Staubli VAL3: findItem.pgx

public program findItem(InstrItem x_iItem, num& x_nResult)
  local num i
  local num l_nSize
  local num j
  local string l_sItem
  local string l_sMessage
  local num l_nResult
  local bool l_bFound
  local InstrItem l_iInstr[3]
  local string l_sSession
begin
  call getSize(l_nSize)
  // scan all the TCP for TCP ON OFF
  for i=0 to l_nSize-1
    call getName(l_sItem,i)
    //
    // SHOW THE TCP name
    //
    call saveData:getSession(l_sSession)
    l_sMessage="TCP "+l_sItem
    call use:typeLen(1,5,l_sMessage,38)
    call getInstr(l_iInstr,true,i)
    // scan deeper for all the action
    for j=0 to size(l_iInstr)-1
      // look inside
      l_bFound=(l_iInstr[j].sType==x_iItem.sType and(l_iInstr[j].sData==x_iItem.sData or find(l_iInstr[j].sData,x_iItem.sData+">")!=-1))
      // use nested items
      l_bFound=l_bFound or find(l_iInstr[j].sType+" "+l_iInstr[j].sData,x_iItem.sData+">")!=-1
      // FOUND IT
      if l_bFound
        x_nResult=-1
        call language:message(l_sMessage,23)
        popUpMsg(l_sMessage+x_iItem.sType+" "+x_iItem.sData+chr(10)+"TCP ON > "+l_iInstr[j].sType+" "+l_iInstr[j].sData)
        // back
        return
      endIf
    endFor
    call getInstr(l_iInstr,false,i)
    // scan deeper for all the action
    for j=0 to size(l_iInstr)-1
      // look inside
      l_bFound=(l_iInstr[j].sType==x_iItem.sType and find(l_iInstr[j].sData,x_iItem.sData)!=-1)
      // FOUND IT
      if l_bFound
        x_nResult=-1
        call language:message(l_sMessage,23)
        popUpMsg(l_sMessage+x_iItem.sType+" "+x_iItem.sData+chr(10)+"TCP OFF > "+l_sItem+" > "+l_iInstr[j].sType+" "+l_iInstr[j].sData)
        // back
        return
      endIf
    endFor
  endFor
end
